{attribute 'linkalways'} 
{attribute 'no_explicit_call' := 'This FB is a CLASS and must be accessed using methods or properties'}
{attribute 'enable_dynamic_creation'}
FUNCTION_BLOCK ABSTRACT KeyValueCollectionEvent EXTENDS Disposable
VAR
	_target : I_KeyValueCollection;
END_VAR

METHOD FB_init : BOOL
VAR_INPUT
	bInitRetains : BOOL; // if TRUE, the retain variables are initialized (warm start / cold start)
	bInCopyCode : BOOL;  // if TRUE, the instance afterwards gets moved into the copy code (online change)
	Target : I_KeyValueCollection;
END_VAR
This^._target := Target;
END_METHOD

PROPERTY PUBLIC Target : I_KeyValueCollection
GET // PUBLIC
Target := _target;
END_GET
END_PROPERTY

END_FUNCTION_BLOCK

(* stored: Version 1.1.0.1, ProductVersion 3.1.4024.12
   POU KeyValueCollectionEvent: Id {d69a3e89-2b8c-03cd-27cf-c614783305cb}, SpecialFunc None
   Folder Constructor: Id {3bef7874-f7f3-054e-3888-91d2f2c6676e}
   Method FB_init: Id {3ef9d006-f969-0ede-0654-0f80a93e3e7b}
   Property Target: Id {fba2f771-7f85-0acd-133a-9fb39e5e31ee}
   Get Get: Id {8ff579e9-703a-0b9c-1c14-8c6d11658c31} *)
